# EPICS substitutions: motorSimApp/Db/sensor.substitutions
file "db/sensor.db"
{

pattern
{P,		N,  M,	MEAN}
{test, 1, m1, 	1.5}
{test, 2, m2, 	0.5}
{test, 3, m3,  -0.5}
{test, 4, m4,  -1.5}
{test, 5, m5,  -2.5}
{test, 6, m6,  -1.0}

}
